FUNCTION_BLOCK INTERNAL FB_DummyModule EXTENDS Fb_ModuleBase
VAR_INPUT
	// Inputs for testing module <> system interaction
	bAllowInit 		: BOOL;
	bAllowAutomatic : BOOL;
	bAllowSemiAuto 	: BOOL;
	bAllowHold 		: BOOL;
	bAllowHome 		: BOOL;
	bAllowReset 	: BOOL;
	bAllowIsSafe 	: BOOL;
	bAllowManual 	: BOOL;
END_VAR
VAR
	nCallsToExecAutomatic : ULINT;
	nCallsToExecHold : ULINT;
	nCallsToExecHome : ULINT;
	nCallsToExecInit : ULINT;
	nCallsToExecManual : ULINT;
	nCallsToExecReset : ULINT;
	nCallsToExecSafeStop : ULINT;
	nCallsToExecSemiAuto : ULINT;
END_VAR

SUPER^();

METHOD PROTECTED  CallComponents : BOOL
VAR_INPUT
END_VAR
END_METHOD

METHOD PROTECTED  CheckCollision : BOOL // Checks device commands for positble collisions  and block if necesarry
VAR_INPUT
END_VAR
END_METHOD

METHOD PROTECTED  ExecAutomatic : BOOL
VAR_INPUT
END_VAR
bAutomatic := bAllowAutomatic;
ExecAutomatic := bAutomatic;

nCallsToExecAutomatic := nCallsToExecAutomatic + 1;
END_METHOD

METHOD PROTECTED  ExecBaseFunctions : BOOL
VAR_INPUT
END_VAR
END_METHOD

METHOD PROTECTED  ExecHold : BOOL
VAR_INPUT
END_VAR
bHeld := bAllowHold;
ExecHold := bHeld;

nCallsToExecHold := nCallsToExecHold + 1;
END_METHOD

METHOD PROTECTED  ExecHome : BOOL
VAR_INPUT
END_VAR
bHomed := bAllowHome;
ExecHome := bHomed;

nCallsToExecHome := nCallsToExecHome + 1;
END_METHOD

METHOD PROTECTED  ExecIdle
VAR_INPUT
END_VAR
END_METHOD

METHOD PROTECTED  ExecInit : BOOL
VAR_INPUT
END_VAR
bInitialized := bAllowInit;
ExecInit := bInitialized;

nCallsToExecInit := nCallsToExecInit + 1;
END_METHOD

METHOD PROTECTED ExecManual : BOOL
VAR_INPUT
END_VAR
bManual := bAllowManual;

nCallsToExecManual := nCallsToExecManual + 1;
END_METHOD

METHOD PROTECTED  ExecReset : BOOL
VAR_INPUT
END_VAR
bResetDone := bAllowReset;
ExecReset := bResetDone;

nCallsToExecReset := nCallsToExecReset + 1;
END_METHOD

METHOD PROTECTED  ExecSafeStop : BOOL
VAR_INPUT
END_VAR
bIsSafe := bAllowIsSafe;
ExecSafeStop := bIsSafe;

nCallsToExecSafeStop := nCallsToExecSafeStop + 1;
END_METHOD

METHOD PROTECTED  ExecSemiAuto : BOOL
VAR_INPUT
END_VAR
bSemiAuto := bAllowSemiAuto;
ExecSemiAuto := bSemiAuto;

nCallsToExecSemiAuto := nCallsToExecSemiAuto + 1;
END_METHOD

END_FUNCTION_BLOCK

(* stored: Version 1.1.0.1, ProductVersion 3.1.4024.11
   POU FB_DummyModule: Id {dcc4cad9-3fe5-4429-9581-93b560acb380}, SpecialFunc None
   Method CallComponents: Id {d2169844-dc1c-4e3e-913f-09fb324d2664}
   Method CheckCollision: Id {4937cc26-00d6-4f3c-bf40-11e88c8d667c}
   Method ExecAutomatic: Id {f8987ceb-7700-4d0d-85e4-b978cef3372f}
   Method ExecBaseFunctions: Id {91fad65e-de57-0ad4-0ec6-0aa0fc0eaaa9}
   Method ExecHold: Id {6ab5aac9-fc82-4cd6-bf01-8fd5a60b4e40}
   Method ExecHome: Id {aba23217-5a2b-4b12-a81c-f311e2a6942f}
   Method ExecIdle: Id {632a345a-3285-0b20-27dd-9762633eb1c8}
   Method ExecInit: Id {02ca3dd5-4e2d-4a98-bf2f-6e10b13580f5}
   Method ExecManual: Id {03354aee-d458-05a7-192c-f10c12f51ba3}
   Method ExecReset: Id {0c5dc2f5-3abd-4b9c-9ed5-e997d45d1f61}
   Method ExecSafeStop: Id {0c490a3e-95f9-4c45-b60a-0f3b24f8a06a}
   Method ExecSemiAuto: Id {bf50ce99-8fec-4331-bd2e-6977f0dad560} *)
